// TIA Portal V18 export
DATA_BLOCK "nokButtonMain_DB"   // DB15
VERSION : 0.1
// stored: AutoNumber true, DBAccessibleFromOPCUA true, DBAccessibleFromWebserver true, InstanceOfName nokButtonMain, InstanceOfType FB
"nokButtonMain"
   // VAR
   //    nokButton1 { S7_SetPoint := 'True'} : "nokButton";
   //    nokButton2 { S7_SetPoint := 'True'} : "nokButton";
   //    nokButtonQUE_Instance { S7_SetPoint := 'True'} : "nokButtonQUE";
   // END_VAR
BEGIN
END_DATA_BLOCK
